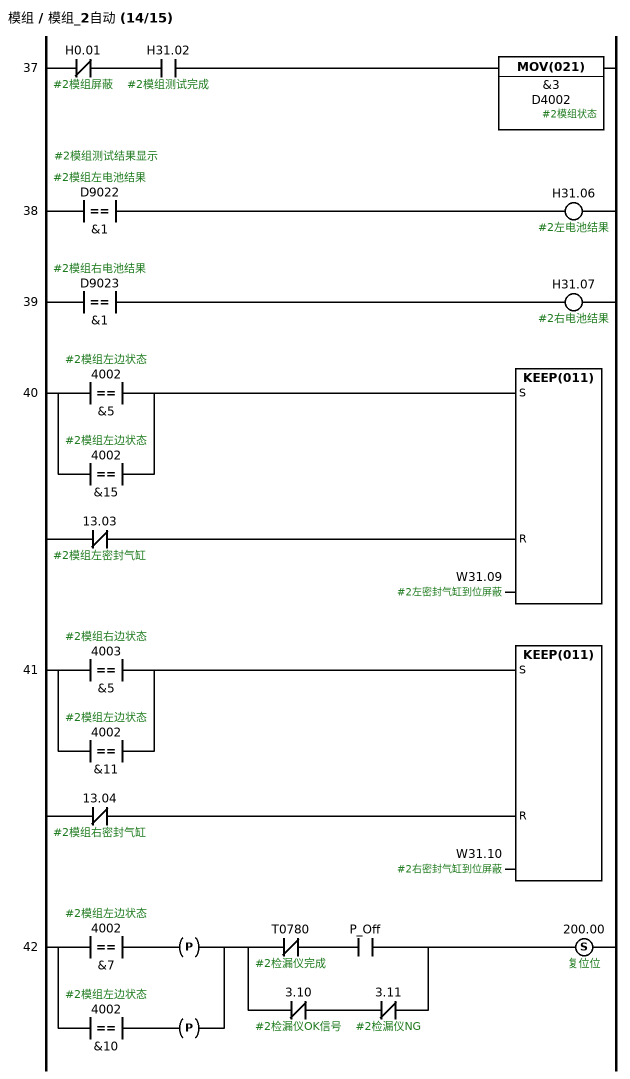
; [picture p233: 模组 / 模组_2自动, rungs 37-42]
; rung 37
LDNOT H0.01  ; #2模组屏蔽
AND H31.02  ; #2模组测试完成
MOV(021) &3 D4002  ; #2模组状态
; rung 38: #2模组测试结果显示
LD=(300) D9022 &1  ; #2模组左电池结果
OUT H31.06  ; #2左电池结果
; rung 39
LD=(300) D9023 &1  ; #2模组右电池结果
OUT H31.07  ; #2右电池结果
; rung 40
LD=(300) 4002 &5  ; #2模组左边状态
OR=(300) 4002 &15  ; #2模组左边状态
LDNOT 13.03  ; #2模组左密封气缸
KEEP(011) W31.09  ; #2左密封气缸到位屏蔽
; rung 41
LD=(300) 4003 &5  ; #2模组右边状态
OR=(300) 4002 &11  ; #2模组左边状态
LDNOT 13.04  ; #2模组右密封气缸
KEEP(011) W31.10  ; #2右密封气缸到位屏蔽
; rung 42
LD=(300) 4002 &7  ; #2模组左边状态
UP(521)
LD=(300) 4002 &10  ; #2模组左边状态
UP(521)
ORLD
LDNOT T0780  ; #2检漏仪完成
AND P_Off
LDNOT 3.10  ; #2检漏仪OK信号  // 2018/5/29hy修改,所有模组不在临抽气结束状态下，测试模组测试完成后，给出停止测试信号
ANDNOT 3.11  ; #2检漏仪NG
ORLD
ANDLD
SET 200.00  ; 复位位

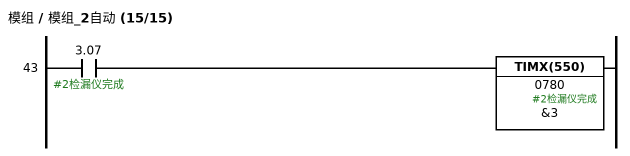
; rung 43
LD 3.07  ; #2检漏仪完成
TIMX(550) 0780 &3  ; #2检漏仪完成

### Section 模组_3自动

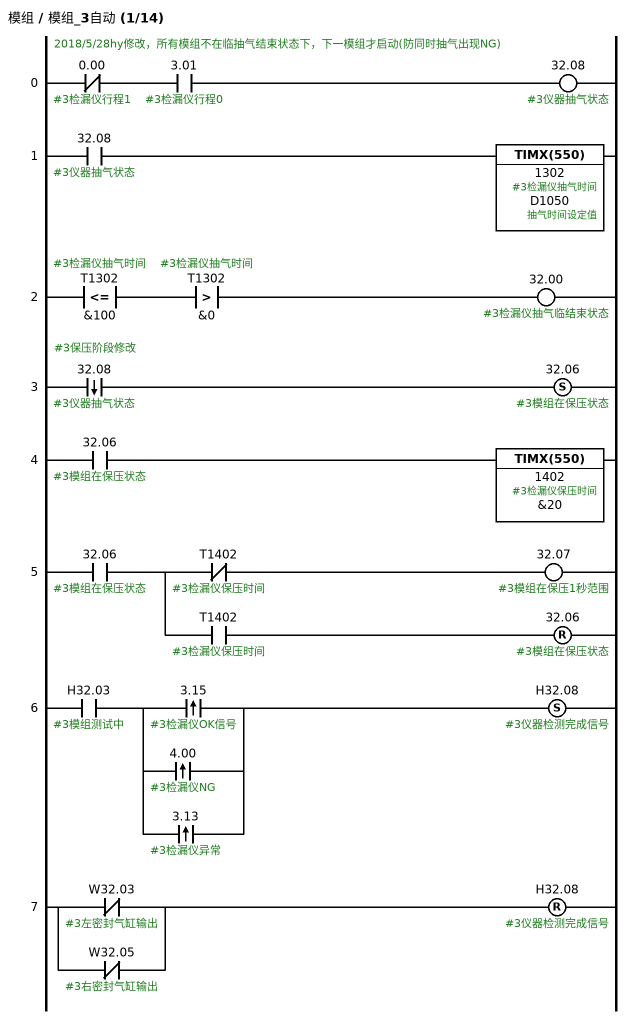
; rung 0: 2018/5/28hy修改，所有模组不在临抽气结束状态下，下一模组才启动(防同时抽气出现NG)
LDNOT 0.00  ; #3检漏仪行程1
AND 3.01  ; #3检漏仪行程0
OUT 32.08  ; #3仪器抽气状态
; rung 1
LD 32.08  ; #3仪器抽气状态
TIMX(550) 1302 D1050  ; 抽气时间设定值, #3检漏仪抽气时间
; rung 2
LD<=(315) T1302 &100  ; #3检漏仪抽气时间
AND>(320) T1302 &0  ; #3检漏仪抽气时间
OUT 32.00  ; #3检漏仪抽气临结束状态
; rung 3: #3保压阶段修改
%LD 32.08  ; #3仪器抽气状态
SET 32.06  ; #3模组在保压状态
; rung 4
LD 32.06  ; #3模组在保压状态
TIMX(550) 1402 &20  ; #3检漏仪保压时间
; rung 5
LD 32.06  ; #3模组在保压状态
OUT TR0
ANDNOT T1402  ; #3检漏仪保压时间
OUT 32.07  ; #3模组在保压1秒范围
LD TR0
AND T1402  ; #3检漏仪保压时间
RSET 32.06  ; #3模组在保压状态
; rung 6
LD H32.03  ; #3模组测试中
@LD 3.15  ; #3检漏仪OK信号
@OR 4.00  ; #3检漏仪NG
@OR 3.13  ; #3检漏仪异常
ANDLD
SET H32.08  ; #3仪器检测完成信号
; rung 7
LDNOT W32.03  ; #3左密封气缸输出
ORNOT W32.05  ; #3右密封气缸输出
RSET H32.08  ; #3仪器检测完成信号

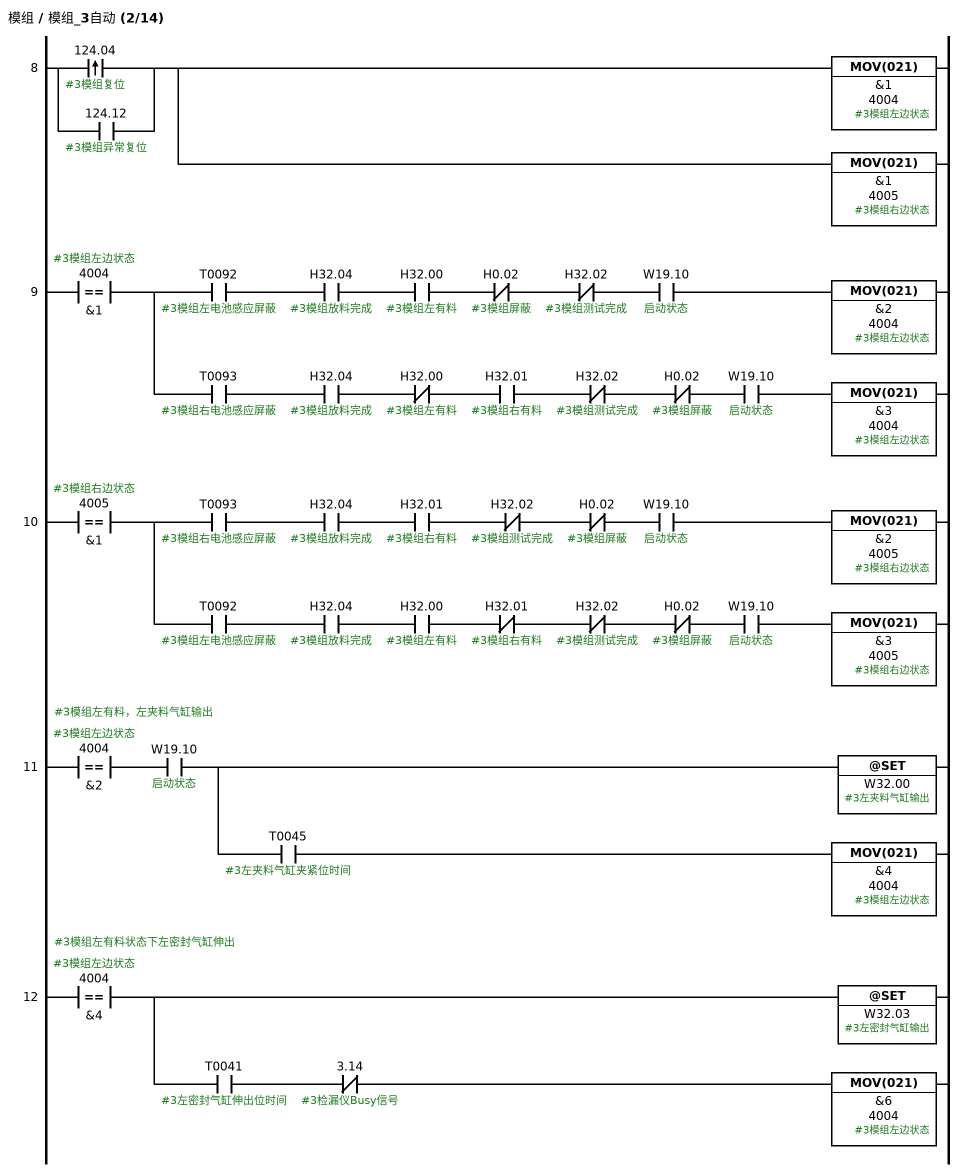
; rung 8
@LD 124.04  ; #3模组复位
OR 124.12  ; #3模组异常复位
MOV(021) &1 4004  ; #3模组左边状态
MOV(021) &1 4005  ; #3模组右边状态
; rung 9
LD=(300) 4004 &1  ; #3模组左边状态
OUT TR0
AND T0092  ; #3模组左电池感应屏蔽
AND H32.04  ; #3模组放料完成
AND H32.00  ; #3模组左有料
ANDNOT H0.02  ; #3模组屏蔽
ANDNOT H32.02  ; #3模组测试完成
AND W19.10  ; 启动状态
MOV(021) &2 4004  ; #3模组左边状态
LD TR0
AND T0093  ; #3模组右电池感应屏蔽
AND H32.04  ; #3模组放料完成
ANDNOT H32.00  ; #3模组左有料
AND H32.01  ; #3模组右有料
ANDNOT H32.02  ; #3模组测试完成
ANDNOT H0.02  ; #3模组屏蔽
AND W19.10  ; 启动状态
MOV(021) &3 4004  ; #3模组左边状态
; rung 10
LD=(300) 4005 &1  ; #3模组右边状态
OUT TR0
AND T0093  ; #3模组右电池感应屏蔽
AND H32.04  ; #3模组放料完成
AND H32.01  ; #3模组右有料
ANDNOT H32.02  ; #3模组测试完成
ANDNOT H0.02  ; #3模组屏蔽
AND W19.10  ; 启动状态
MOV(021) &2 4005  ; #3模组右边状态
LD TR0
AND T0092  ; #3模组左电池感应屏蔽
AND H32.04  ; #3模组放料完成
AND H32.00  ; #3模组左有料
ANDNOT H32.01  ; #3模组右有料
ANDNOT H32.02  ; #3模组测试完成
ANDNOT H0.02  ; #3模组屏蔽
AND W19.10  ; 启动状态
MOV(021) &3 4005  ; #3模组右边状态
; rung 11: #3模组左有料，左夹料气缸输出
LD=(300) 4004 &2  ; #3模组左边状态
AND W19.10  ; 启动状态
@SET W32.00  ; #3左夹料气缸输出
AND T0045  ; #3左夹料气缸夹紧位时间
MOV(021) &4 4004  ; #3模组左边状态
; rung 12: #3模组左有料状态下左密封气缸伸出
LD=(300) 4004 &4  ; #3模组左边状态
@SET W32.03  ; #3左密封气缸输出
AND T0041  ; #3左密封气缸伸出位时间
ANDNOT 3.14  ; #3检漏仪Busy信号
MOV(021) &6 4004  ; #3模组左边状态

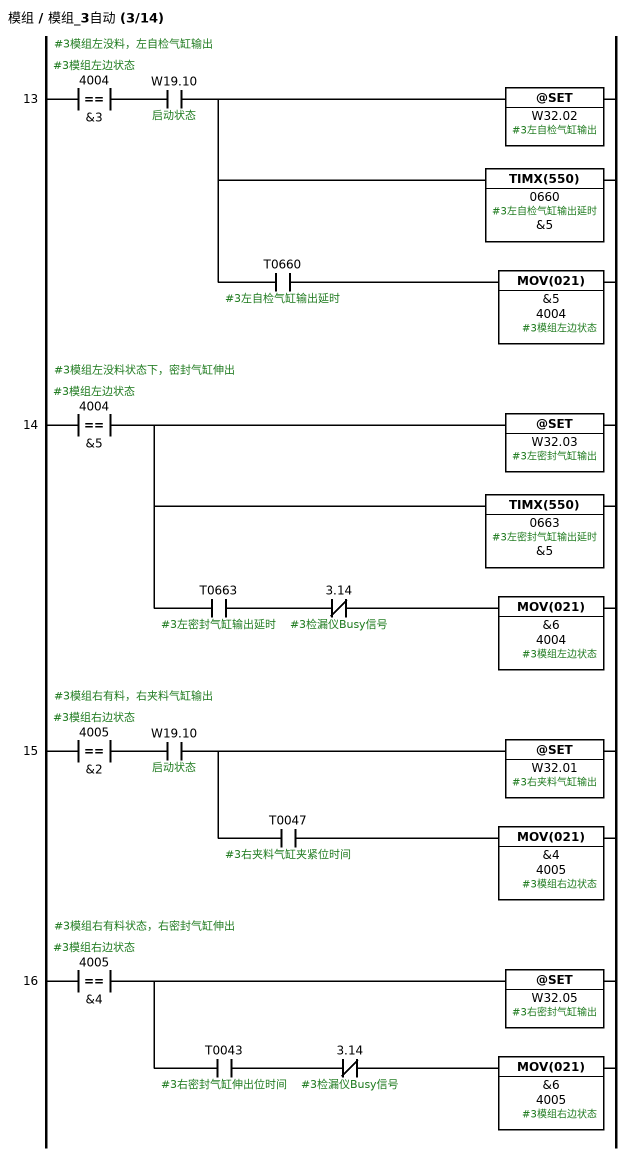
; rung 13: #3模组左没料，左自检气缸输出
LD=(300) 4004 &3  ; #3模组左边状态
AND W19.10  ; 启动状态
@SET W32.02  ; #3左自检气缸输出
TIMX(550) 0660 &5  ; #3左自检气缸输出延时
AND T0660  ; #3左自检气缸输出延时
MOV(021) &5 4004  ; #3模组左边状态
; rung 14: #3模组左没料状态下，密封气缸伸出
LD=(300) 4004 &5  ; #3模组左边状态
@SET W32.03  ; #3左密封气缸输出
TIMX(550) 0663 &5  ; #3左密封气缸输出延时
AND T0663  ; #3左密封气缸输出延时
ANDNOT 3.14  ; #3检漏仪Busy信号
MOV(021) &6 4004  ; #3模组左边状态
; rung 15: #3模组右有料，右夹料气缸输出
LD=(300) 4005 &2  ; #3模组右边状态
AND W19.10  ; 启动状态
@SET W32.01  ; #3右夹料气缸输出
AND T0047  ; #3右夹料气缸夹紧位时间
MOV(021) &4 4005  ; #3模组右边状态
; rung 16: #3模组右有料状态，右密封气缸伸出
LD=(300) 4005 &4  ; #3模组右边状态
@SET W32.05  ; #3右密封气缸输出
AND T0043  ; #3右密封气缸伸出位时间
ANDNOT 3.14  ; #3检漏仪Busy信号
MOV(021) &6 4005  ; #3模组右边状态

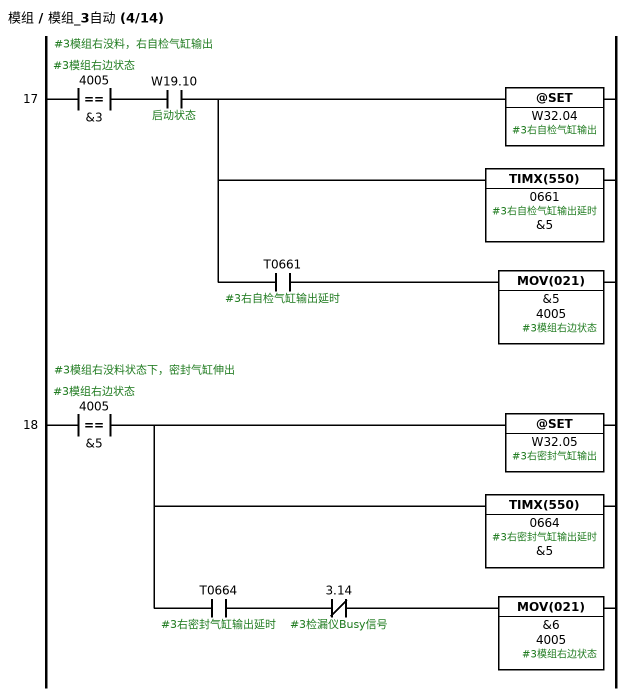
; rung 17: #3模组右没料，右自检气缸输出
LD=(300) 4005 &3  ; #3模组右边状态
AND W19.10  ; 启动状态
@SET W32.04  ; #3右自检气缸输出
TIMX(550) 0661 &5  ; #3右自检气缸输出延时
AND T0661  ; #3右自检气缸输出延时
MOV(021) &5 4005  ; #3模组右边状态
; rung 18: #3模组右没料状态下，密封气缸伸出
LD=(300) 4005 &5  ; #3模组右边状态
@SET W32.05  ; #3右密封气缸输出
TIMX(550) 0664 &5  ; #3右密封气缸输出延时
AND T0664  ; #3右密封气缸输出延时
ANDNOT 3.14  ; #3检漏仪Busy信号
MOV(021) &6 4005  ; #3模组右边状态

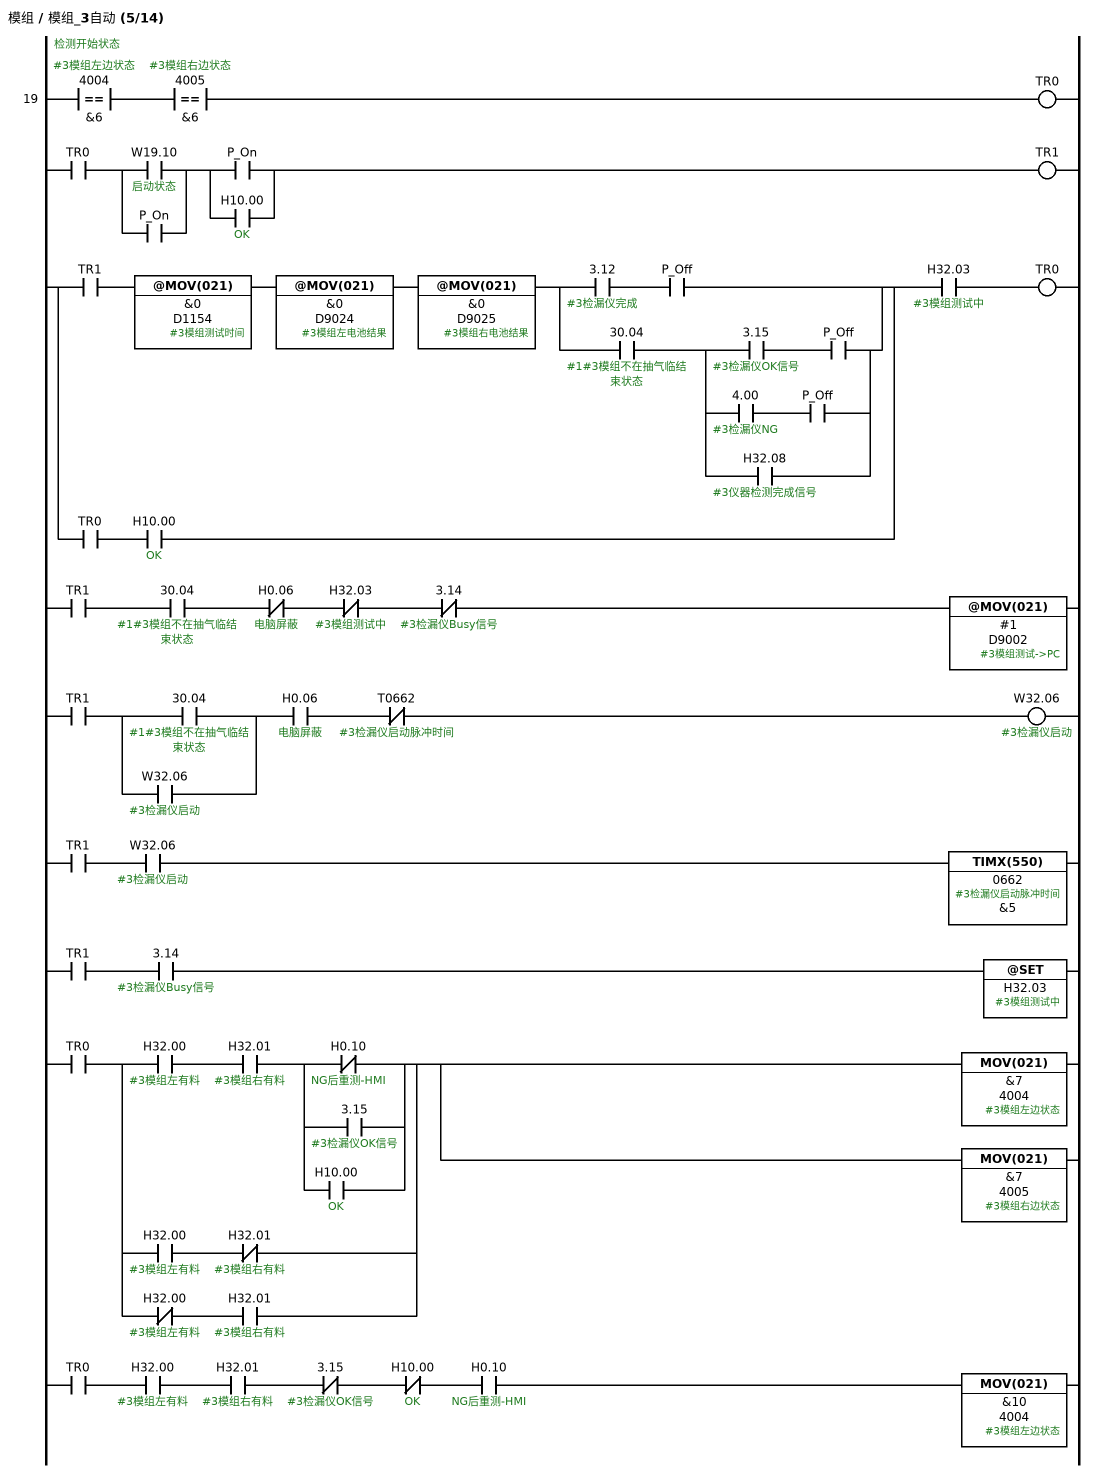
; rung 19: 检测开始状态
LD=(300) 4004 &6  ; #3模组左边状态
AND=(300) 4005 &6  ; #3模组右边状态
OUT TR0
LD W19.10  ; 启动状态
OR P_On
ANDLD
LD P_On  // 2018/5/28hy修改 所有模组不在抽气临结束状态下，下一模组才能启动(防抽气NG)
OR H10.00  ; OK
ANDLD
OUT TR1
AND 30.04  ; #1#3模组不在抽气临结束状态  // 2018/5/28hy修改 所有模组不在抽气临结束状态下，下一模组才能启动(防抽气NG)
ANDNOT H0.06  ; 电脑屏蔽
ANDNOT H32.03  ; #3模组测试中
ANDNOT 3.14  ; #3检漏仪Busy信号
@MOV(021) #1 D9002  ; #3模组测试->PC
LD TR1
LD 30.04  ; #1#3模组不在抽气临结束状态  // 2018/5/28hy修改 所有模组不在抽气临结束状态下，下一模组才能启动(防抽气NG)
OR W32.06  ; #3检漏仪启动
ANDLD
AND H0.06  ; 电脑屏蔽
ANDNOT T0662  ; #3检漏仪启动脉冲时间
OUT W32.06  ; #3检漏仪启动
LD TR1
AND W32.06  ; #3检漏仪启动
TIMX(550) 0662 &5  ; #3检漏仪启动脉冲时间
LD TR1
AND 3.14  ; #3检漏仪Busy信号
@SET H32.03  ; #3模组测试中
LD TR1
@MOV(021) &0 D1154  ; #3模组测试时间
@MOV(021) &0 D9024  ; #3模组左电池结果
@MOV(021) &0 D9025  ; #3模组右电池结果
LD 3.12  ; #3检漏仪完成
AND P_Off
LD 30.04  ; #1#3模组不在抽气临结束状态  // 2018/5/29hy修改,所有模组不在临抽气结束状态下，测试模组测试完成后，给出停止测试信号
LD 3.15  ; #3检漏仪OK信号
AND P_Off
LD 4.00  ; #3检漏仪NG
AND P_Off
ORLD
OR H32.08  ; #3仪器检测完成信号
ANDLD
ORLD
ANDLD
LD TR0
AND H10.00  ; OK
ORLD
AND H32.03  ; #3模组测试中
OUT TR0
LD H32.00  ; #3模组左有料
AND H32.01  ; #3模组右有料
LDNOT H0.10  ; NG后重测-HMI
OR 3.15  ; #3检漏仪OK信号
OR H10.00  ; OK
ANDLD
LD H32.00  ; #3模组左有料
ANDNOT H32.01  ; #3模组右有料
ORLD
LDNOT H32.00  ; #3模组左有料
AND H32.01  ; #3模组右有料
ORLD
ANDLD
MOV(021) &7 4004  ; #3模组左边状态
MOV(021) &7 4005  ; #3模组右边状态
LD TR0
AND H32.00  ; #3模组左有料
AND H32.01  ; #3模组右有料
ANDNOT 3.15  ; #3检漏仪OK信号
ANDNOT H10.00  ; OK
AND H0.10  ; NG后重测-HMI
MOV(021) &10 4004  ; #3模组左边状态

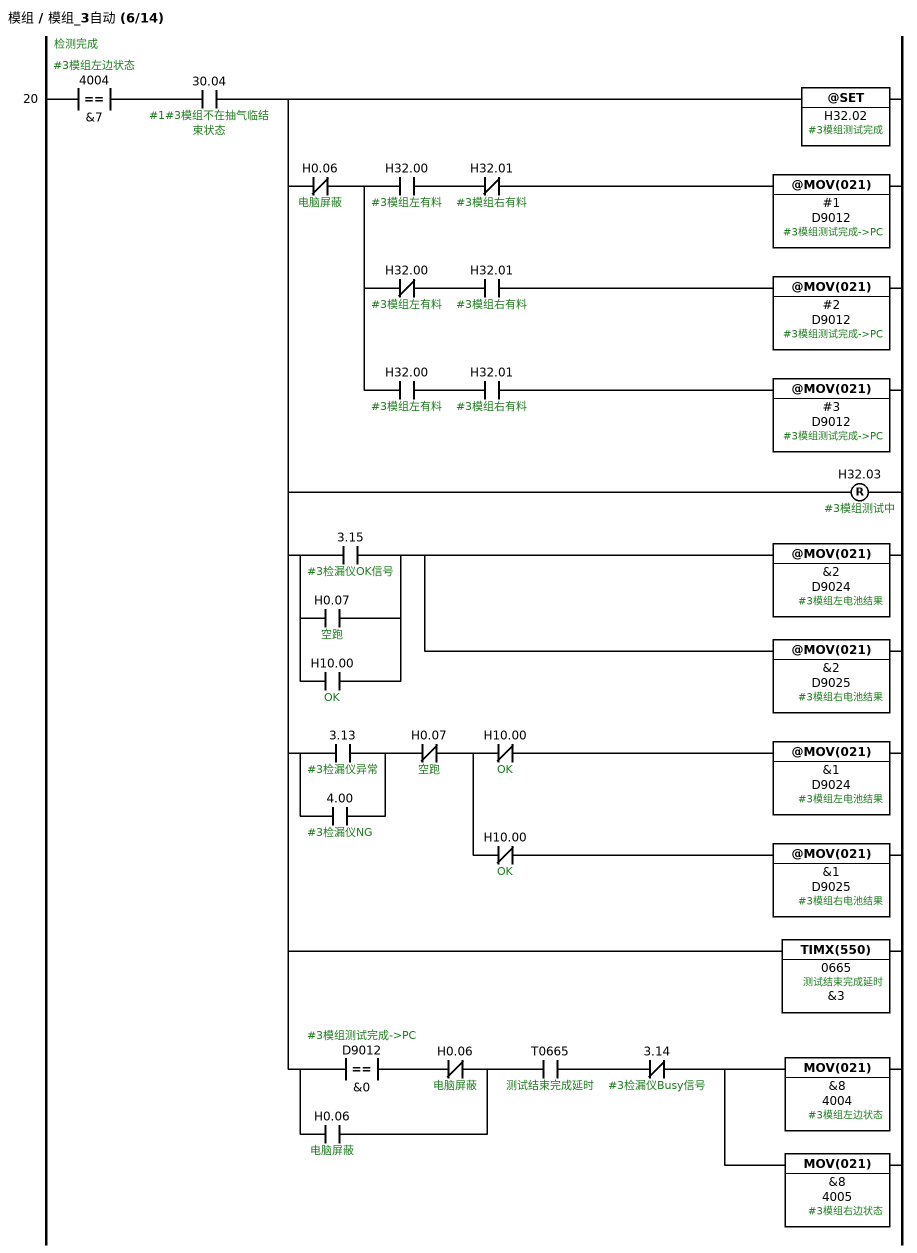
; rung 20: 检测完成
LD=(300) 4004 &7  ; #3模组左边状态
AND 30.04  ; #1#3模组不在抽气临结束状态
OUT TR0
@SET H32.02  ; #3模组测试完成
ANDNOT H0.06  ; 电脑屏蔽
OUT TR1
AND H32.00  ; #3模组左有料
ANDNOT H32.01  ; #3模组右有料
@MOV(021) #1 D9012  ; #3模组测试完成->PC
LD TR1
ANDNOT H32.00  ; #3模组左有料
AND H32.01  ; #3模组右有料
@MOV(021) #2 D9012  ; #3模组测试完成->PC
LD TR1
AND H32.00  ; #3模组左有料
AND H32.01  ; #3模组右有料
@MOV(021) #3 D9012  ; #3模组测试完成->PC
LD TR0
RSET H32.03  ; #3模组测试中
LD 3.15  ; #3检漏仪OK信号
OR H0.07  ; 空跑
OR H10.00  ; OK
ANDLD
@MOV(021) &2 D9024  ; #3模组左电池结果
@MOV(021) &2 D9025  ; #3模组右电池结果
LD TR0
LD 3.13  ; #3检漏仪异常
OR 4.00  ; #3检漏仪NG
ANDLD
ANDNOT H0.07  ; 空跑
OUT TR1
ANDNOT H10.00  ; OK
@MOV(021) &1 D9024  ; #3模组左电池结果
LD TR1
ANDNOT H10.00  ; OK
@MOV(021) &1 D9025  ; #3模组右电池结果
LD TR0
TIMX(550) 0665 &3  ; 测试结束完成延时
LD=(300) D9012 &0  ; #3模组测试完成->PC
ANDNOT H0.06  ; 电脑屏蔽
OR H0.06  ; 电脑屏蔽
ANDLD
AND T0665  ; 测试结束完成延时
ANDNOT 3.14  ; #3检漏仪Busy信号
MOV(021) &8 4004  ; #3模组左边状态
MOV(021) &8 4005  ; #3模组右边状态

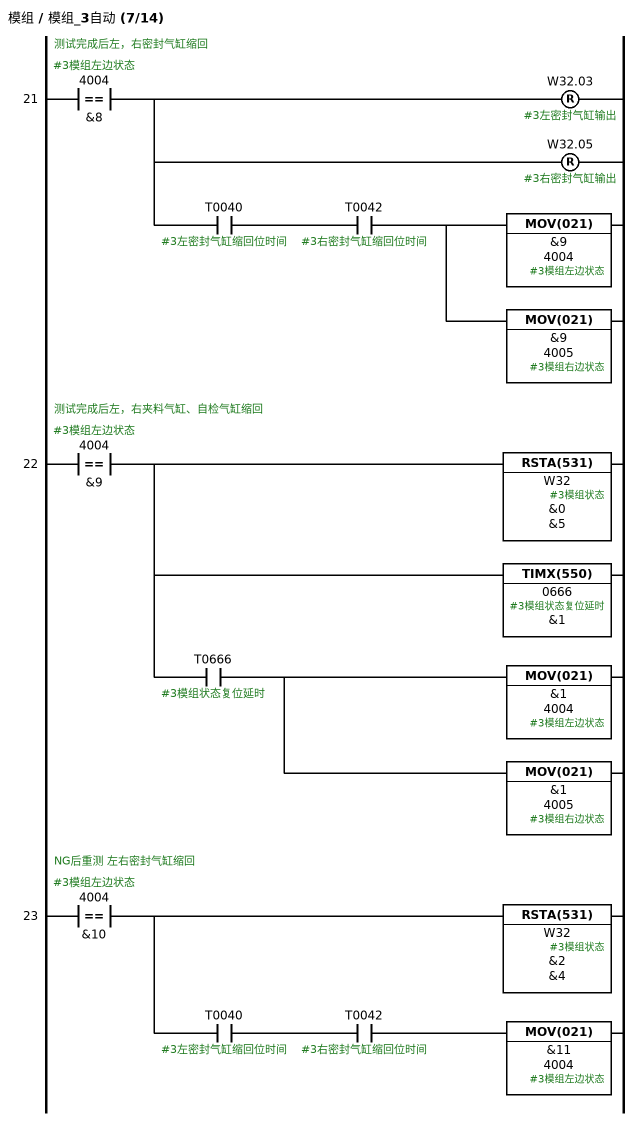
; rung 21: 测试完成后左，右密封气缸缩回
LD=(300) 4004 &8  ; #3模组左边状态
RSET W32.03  ; #3左密封气缸输出
RSET W32.05  ; #3右密封气缸输出
AND T0040  ; #3左密封气缸缩回位时间
AND T0042  ; #3右密封气缸缩回位时间
MOV(021) &9 4004  ; #3模组左边状态
MOV(021) &9 4005  ; #3模组右边状态
; rung 22: 测试完成后左，右夹料气缸、自检气缸缩回
LD=(300) 4004 &9  ; #3模组左边状态
RSTA(531) W32 &0 &5  ; #3模组状态
TIMX(550) 0666 &1  ; #3模组状态复位延时
AND T0666  ; #3模组状态复位延时
MOV(021) &1 4004  ; #3模组左边状态
MOV(021) &1 4005  ; #3模组右边状态
; rung 23: NG后重测 左右密封气缸缩回
LD=(300) 4004 &10  ; #3模组左边状态
RSTA(531) W32 &2 &4  ; #3模组状态
AND T0040  ; #3左密封气缸缩回位时间
AND T0042  ; #3右密封气缸缩回位时间
MOV(021) &11 4004  ; #3模组左边状态

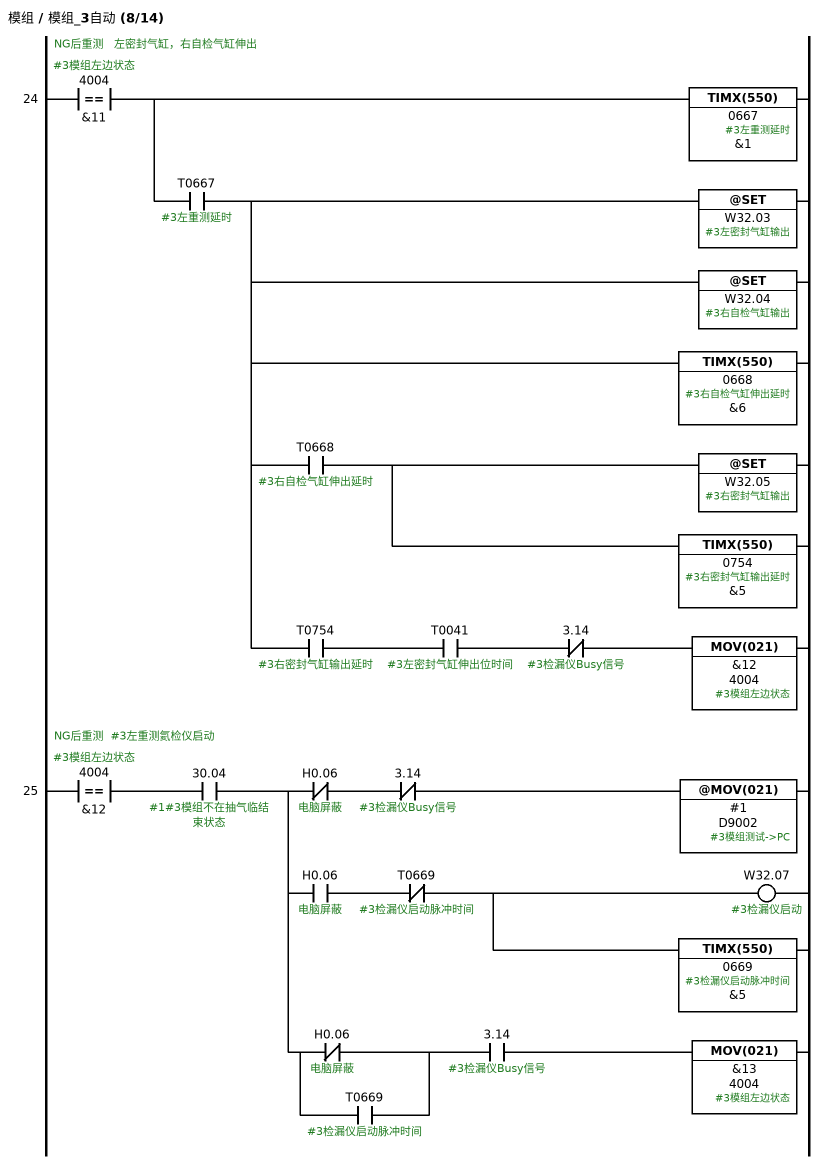
; rung 24: NG后重测   左密封气缸，右自检气缸伸出
LD=(300) 4004 &11  ; #3模组左边状态
TIMX(550) 0667 &1  ; #3左重测延时
AND T0667  ; #3左重测延时
OUT TR0
@SET W32.03  ; #3左密封气缸输出
@SET W32.04  ; #3右自检气缸输出
TIMX(550) 0668 &6  ; #3右自检气缸伸出延时
AND T0668  ; #3右自检气缸伸出延时
@SET W32.05  ; #3右密封气缸输出
TIMX(550) 0754 &5  ; #3右密封气缸输出延时
LD TR0
AND T0754  ; #3右密封气缸输出延时
AND T0041  ; #3左密封气缸伸出位时间
ANDNOT 3.14  ; #3检漏仪Busy信号
MOV(021) &12 4004  ; #3模组左边状态
; rung 25: NG后重测  #3左重测氦检仪启动
LD=(300) 4004 &12  ; #3模组左边状态
AND 30.04  ; #1#3模组不在抽气临结束状态  // 2018/5/28hy修改 所有模组不在抽气临结束状态下，下一模组才能启动(防抽气NG)
OUT TR0
ANDNOT H0.06  ; 电脑屏蔽
ANDNOT 3.14  ; #3检漏仪Busy信号
@MOV(021) #1 D9002  ; #3模组测试->PC
LD TR0
AND H0.06  ; 电脑屏蔽
ANDNOT T0669  ; #3检漏仪启动脉冲时间
OUT W32.07  ; #3检漏仪启动
TIMX(550) 0669 &5  ; #3检漏仪启动脉冲时间
LD TR0
LDNOT H0.06  ; 电脑屏蔽
OR T0669  ; #3检漏仪启动脉冲时间
ANDLD
AND 3.14  ; #3检漏仪Busy信号
MOV(021) &13 4004  ; #3模组左边状态

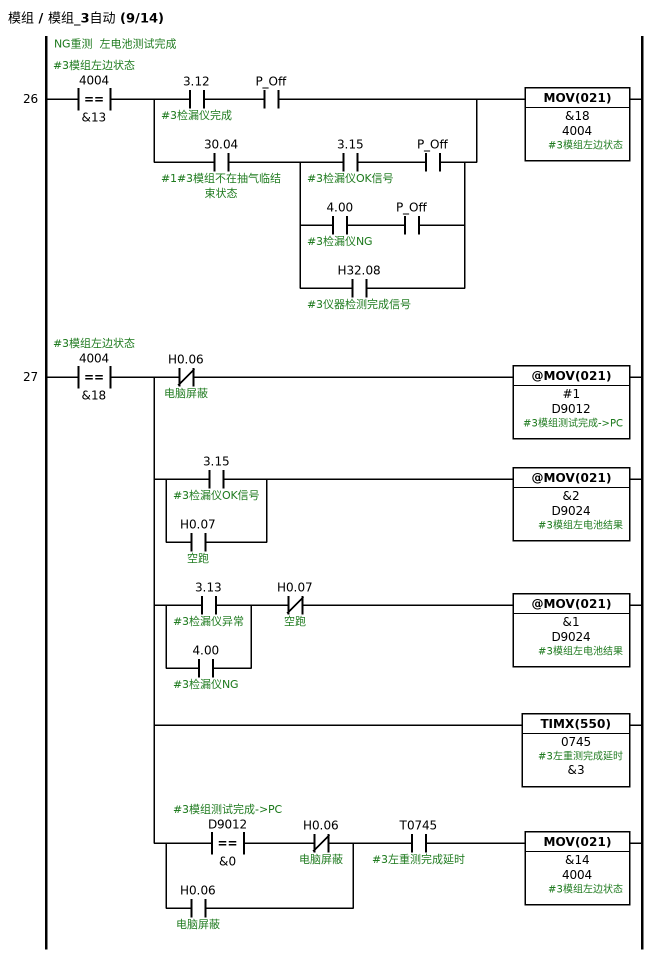
; rung 26: NG重测  左电池测试完成
LD=(300) 4004 &13  ; #3模组左边状态
LD 3.12  ; #3检漏仪完成
AND P_Off
LD 30.04  ; #1#3模组不在抽气临结束状态  // 2018/5/29hy修改,所有模组不在临抽气结束状态下，测试模组测试完成后，给出停止测试信号
LD 3.15  ; #3检漏仪OK信号
AND P_Off
LD 4.00  ; #3检漏仪NG
AND P_Off
ORLD
OR H32.08  ; #3仪器检测完成信号
ANDLD
ORLD
ANDLD
MOV(021) &18 4004  ; #3模组左边状态
; rung 27
LD=(300) 4004 &18  ; #3模组左边状态
OUT TR0
ANDNOT H0.06  ; 电脑屏蔽
@MOV(021) #1 D9012  ; #3模组测试完成->PC
LD TR0
LD 3.15  ; #3检漏仪OK信号
OR H0.07  ; 空跑
ANDLD
@MOV(021) &2 D9024  ; #3模组左电池结果
LD TR0
LD 3.13  ; #3检漏仪异常
OR 4.00  ; #3检漏仪NG
ANDLD
ANDNOT H0.07  ; 空跑
@MOV(021) &1 D9024  ; #3模组左电池结果
LD TR0
TIMX(550) 0745 &3  ; #3左重测完成延时
LD=(300) D9012 &0  ; #3模组测试完成->PC
ANDNOT H0.06  ; 电脑屏蔽
OR H0.06  ; 电脑屏蔽
ANDLD
AND T0745  ; #3左重测完成延时
MOV(021) &14 4004  ; #3模组左边状态

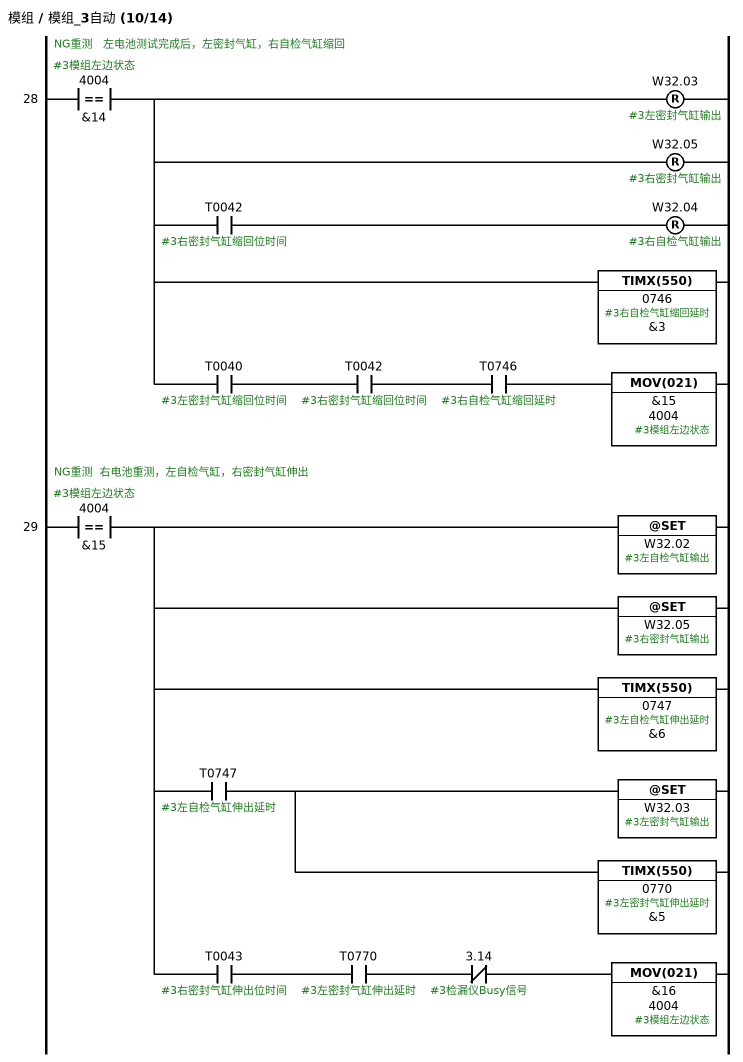
; rung 28: NG重测   左电池测试完成后，左密封气缸，右自检气缸缩回
LD=(300) 4004 &14  ; #3模组左边状态
OUT TR0
RSET W32.03  ; #3左密封气缸输出
RSET W32.05  ; #3右密封气缸输出
AND T0042  ; #3右密封气缸缩回位时间
RSET W32.04  ; #3右自检气缸输出
LD TR0
TIMX(550) 0746 &3  ; #3右自检气缸缩回延时
AND T0040  ; #3左密封气缸缩回位时间
AND T0042  ; #3右密封气缸缩回位时间
AND T0746  ; #3右自检气缸缩回延时
MOV(021) &15 4004  ; #3模组左边状态
; rung 29: NG重测  右电池重测，左自检气缸，右密封气缸伸出
LD=(300) 4004 &15  ; #3模组左边状态
OUT TR0
@SET W32.02  ; #3左自检气缸输出
@SET W32.05  ; #3右密封气缸输出
TIMX(550) 0747 &6  ; #3左自检气缸伸出延时
AND T0747  ; #3左自检气缸伸出延时
@SET W32.03  ; #3左密封气缸输出
TIMX(550) 0770 &5  ; #3左密封气缸伸出延时
LD TR0
AND T0043  ; #3右密封气缸伸出位时间
AND T0770  ; #3左密封气缸伸出延时
ANDNOT 3.14  ; #3检漏仪Busy信号
MOV(021) &16 4004  ; #3模组左边状态

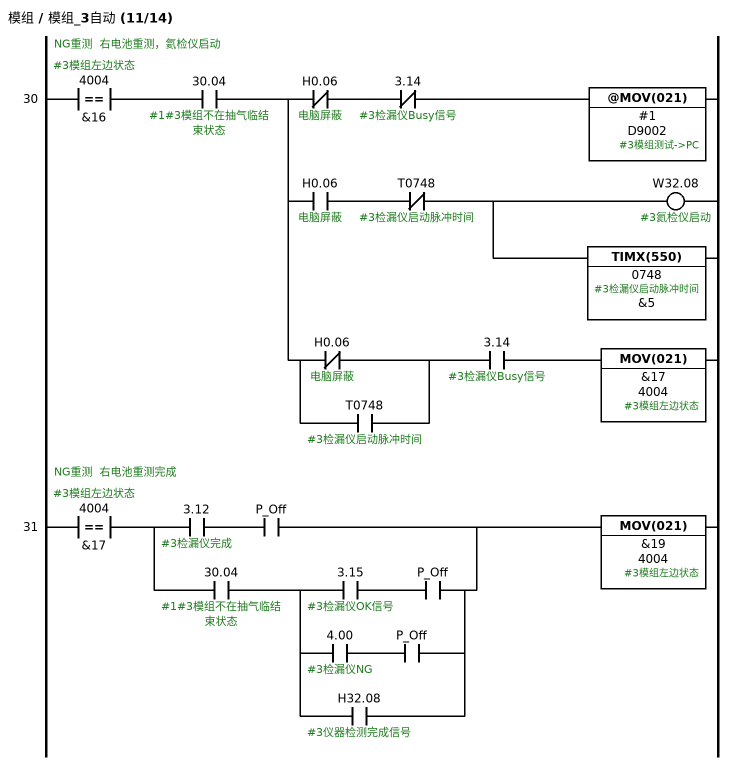
; rung 30: NG重测  右电池重测，氦检仪启动
LD=(300) 4004 &16  ; #3模组左边状态
AND 30.04  ; #1#3模组不在抽气临结束状态  // 2018/5/28hy修改 所有模组不在抽气临结束状态下，下一模组才能启动(防抽气NG)
OUT TR0
ANDNOT H0.06  ; 电脑屏蔽
ANDNOT 3.14  ; #3检漏仪Busy信号
@MOV(021) #1 D9002  ; #3模组测试->PC
LD TR0
AND H0.06  ; 电脑屏蔽
ANDNOT T0748  ; #3检漏仪启动脉冲时间
OUT W32.08  ; #3氦检仪启动
TIMX(550) 0748 &5  ; #3检漏仪启动脉冲时间
LD TR0
LDNOT H0.06  ; 电脑屏蔽
OR T0748  ; #3检漏仪启动脉冲时间
ANDLD
AND 3.14  ; #3检漏仪Busy信号
MOV(021) &17 4004  ; #3模组左边状态
; rung 31: NG重测  右电池重测完成
LD=(300) 4004 &17  ; #3模组左边状态
LD 3.12  ; #3检漏仪完成
AND P_Off
LD 30.04  ; #1#3模组不在抽气临结束状态  // 2018/5/29hy修改,所有模组不在临抽气结束状态下，测试模组测试完成后，给出停止测试信号
LD 3.15  ; #3检漏仪OK信号
AND P_Off
LD 4.00  ; #3检漏仪NG
AND P_Off
ORLD
OR H32.08  ; #3仪器检测完成信号
ANDLD
ORLD
ANDLD
MOV(021) &19 4004  ; #3模组左边状态

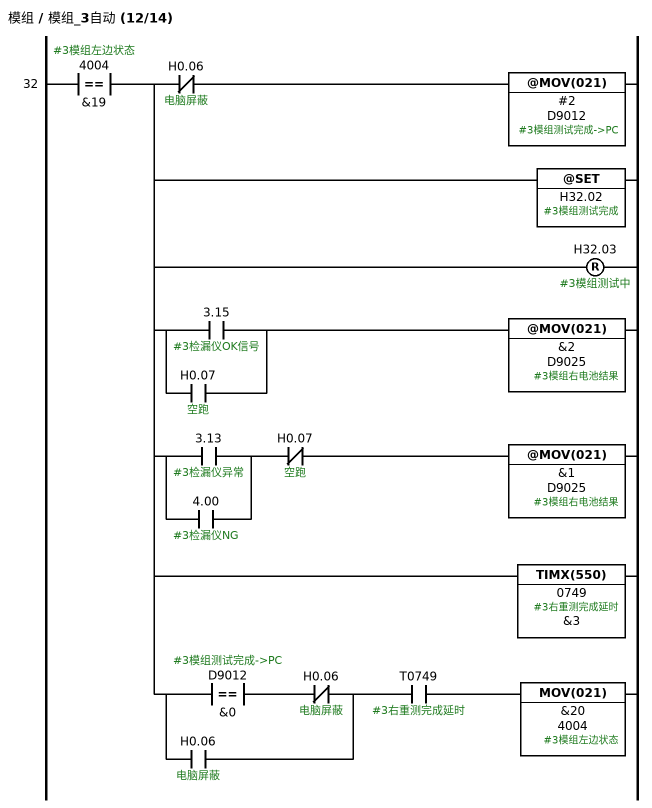
; rung 32
LD=(300) 4004 &19  ; #3模组左边状态
OUT TR0
ANDNOT H0.06  ; 电脑屏蔽
@MOV(021) #2 D9012  ; #3模组测试完成->PC
LD TR0
@SET H32.02  ; #3模组测试完成
RSET H32.03  ; #3模组测试中
LD 3.15  ; #3检漏仪OK信号
OR H0.07  ; 空跑
ANDLD
@MOV(021) &2 D9025  ; #3模组右电池结果
LD TR0
LD 3.13  ; #3检漏仪异常
OR 4.00  ; #3检漏仪NG
ANDLD
ANDNOT H0.07  ; 空跑
@MOV(021) &1 D9025  ; #3模组右电池结果
LD TR0
TIMX(550) 0749 &3  ; #3右重测完成延时
LD=(300) D9012 &0  ; #3模组测试完成->PC
ANDNOT H0.06  ; 电脑屏蔽
OR H0.06  ; 电脑屏蔽
ANDLD
AND T0749  ; #3右重测完成延时
MOV(021) &20 4004  ; #3模组左边状态

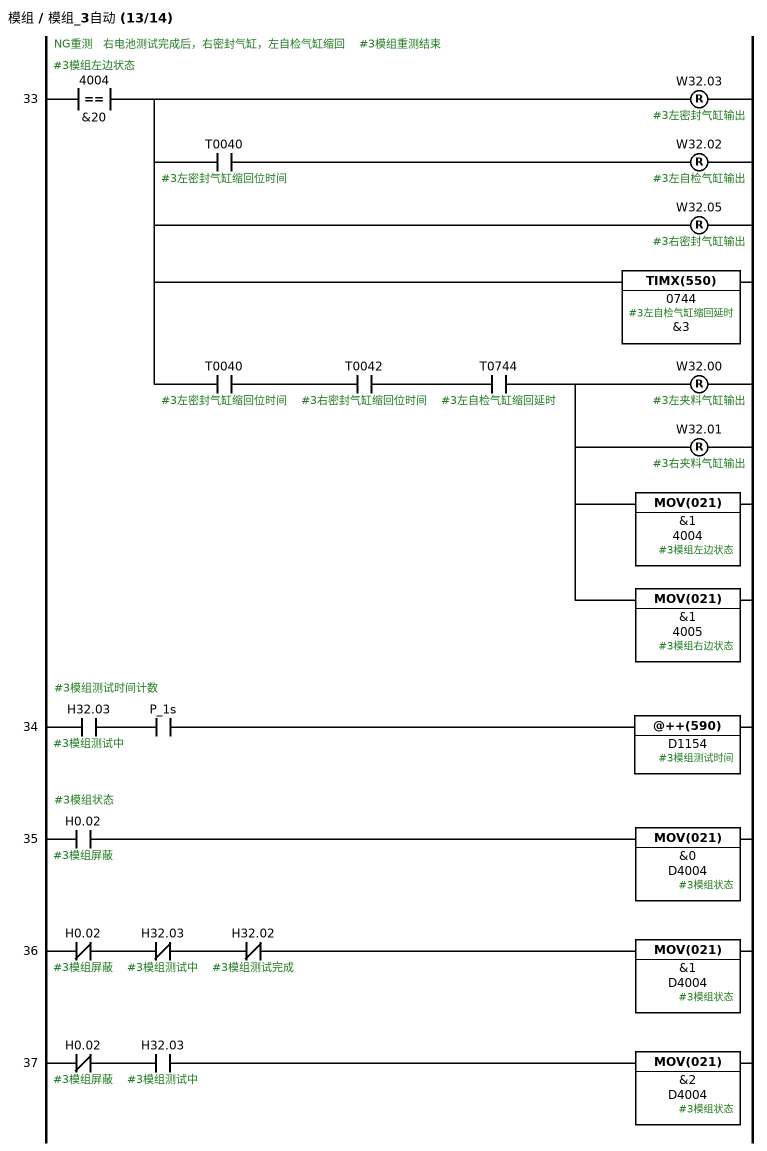
; rung 33: NG重测   右电池测试完成后，右密封气缸，左自检气缸缩回    #3模组重测结束
LD=(300) 4004 &20  ; #3模组左边状态
OUT TR0
RSET W32.03  ; #3左密封气缸输出
AND T0040  ; #3左密封气缸缩回位时间
RSET W32.02  ; #3左自检气缸输出
LD TR0
RSET W32.05  ; #3右密封气缸输出
TIMX(550) 0744 &3  ; #3左自检气缸缩回延时
AND T0040  ; #3左密封气缸缩回位时间
AND T0042  ; #3右密封气缸缩回位时间
AND T0744  ; #3左自检气缸缩回延时
RSET W32.00  ; #3左夹料气缸输出
RSET W32.01  ; #3右夹料气缸输出
MOV(021) &1 4004  ; #3模组左边状态
MOV(021) &1 4005  ; #3模组右边状态
; rung 34: #3模组测试时间计数
LD H32.03  ; #3模组测试中
AND P_1s
@++(590) D1154  ; #3模组测试时间
; rung 35: #3模组状态
LD H0.02  ; #3模组屏蔽
MOV(021) &0 D4004  ; #3模组状态
; rung 36
LDNOT H0.02  ; #3模组屏蔽
ANDNOT H32.03  ; #3模组测试中
ANDNOT H32.02  ; #3模组测试完成
MOV(021) &1 D4004  ; #3模组状态
; rung 37
LDNOT H0.02  ; #3模组屏蔽
AND H32.03  ; #3模组测试中
MOV(021) &2 D4004  ; #3模组状态

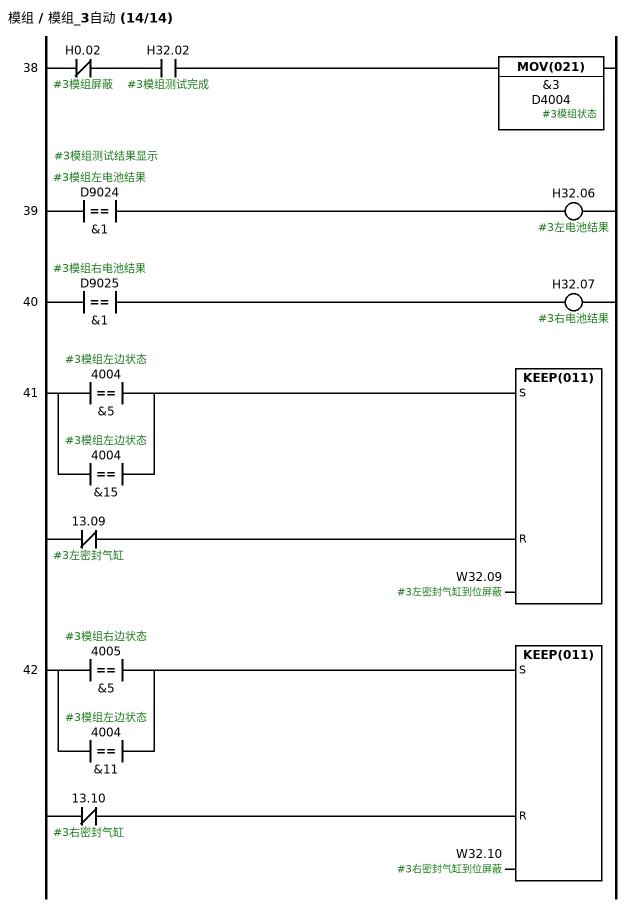
; rung 38
LDNOT H0.02  ; #3模组屏蔽
AND H32.02  ; #3模组测试完成
MOV(021) &3 D4004  ; #3模组状态
; rung 39: #3模组测试结果显示
LD=(300) D9024 &1  ; #3模组左电池结果
OUT H32.06  ; #3左电池结果
; rung 40
LD=(300) D9025 &1  ; #3模组右电池结果
OUT H32.07  ; #3右电池结果
; rung 41
LD=(300) 4004 &5  ; #3模组左边状态
OR=(300) 4004 &15  ; #3模组左边状态
LDNOT 13.09  ; #3左密封气缸
KEEP(011) W32.09  ; #3左密封气缸到位屏蔽
; rung 42
LD=(300) 4005 &5  ; #3模组右边状态
OR=(300) 4004 &11  ; #3模组左边状态
LDNOT 13.10  ; #3右密封气缸
KEEP(011) W32.10  ; #3右密封气缸到位屏蔽

### Section 模组_4自动

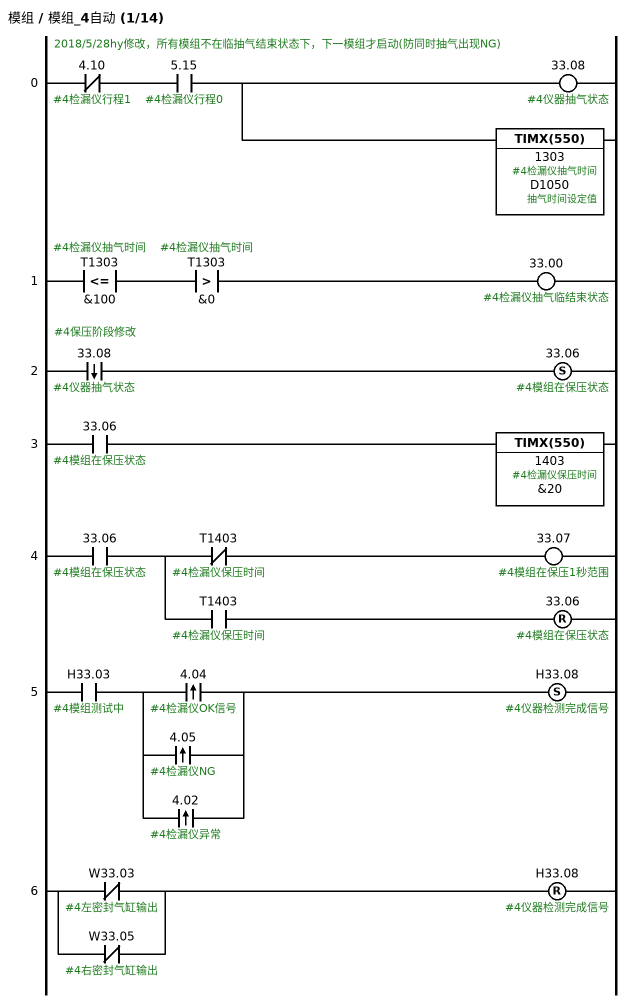
; rung 0: 2018/5/28hy修改，所有模组不在临抽气结束状态下，下一模组才启动(防同时抽气出现NG)
LDNOT 4.10  ; #4检漏仪行程1
AND 5.15  ; #4检漏仪行程0
OUT 33.08  ; #4仪器抽气状态
TIMX(550) 1303 D1050  ; 抽气时间设定值, #4检漏仪抽气时间
; rung 1
LD<=(315) T1303 &100  ; #4检漏仪抽气时间
AND>(320) T1303 &0  ; #4检漏仪抽气时间
OUT 33.00  ; #4检漏仪抽气临结束状态
; rung 2: #4保压阶段修改
%LD 33.08  ; #4仪器抽气状态
SET 33.06  ; #4模组在保压状态
; rung 3
LD 33.06  ; #4模组在保压状态
TIMX(550) 1403 &20  ; #4检漏仪保压时间
; rung 4
LD 33.06  ; #4模组在保压状态
OUT TR0
ANDNOT T1403  ; #4检漏仪保压时间
OUT 33.07  ; #4模组在保压1秒范围
LD TR0
AND T1403  ; #4检漏仪保压时间
RSET 33.06  ; #4模组在保压状态
; rung 5
LD H33.03  ; #4模组测试中
@LD 4.04  ; #4检漏仪OK信号
@OR 4.05  ; #4检漏仪NG
@OR 4.02  ; #4检漏仪异常
ANDLD
SET H33.08  ; #4仪器检测完成信号
; rung 6
LDNOT W33.03  ; #4左密封气缸输出
ORNOT W33.05  ; #4右密封气缸输出
RSET H33.08  ; #4仪器检测完成信号

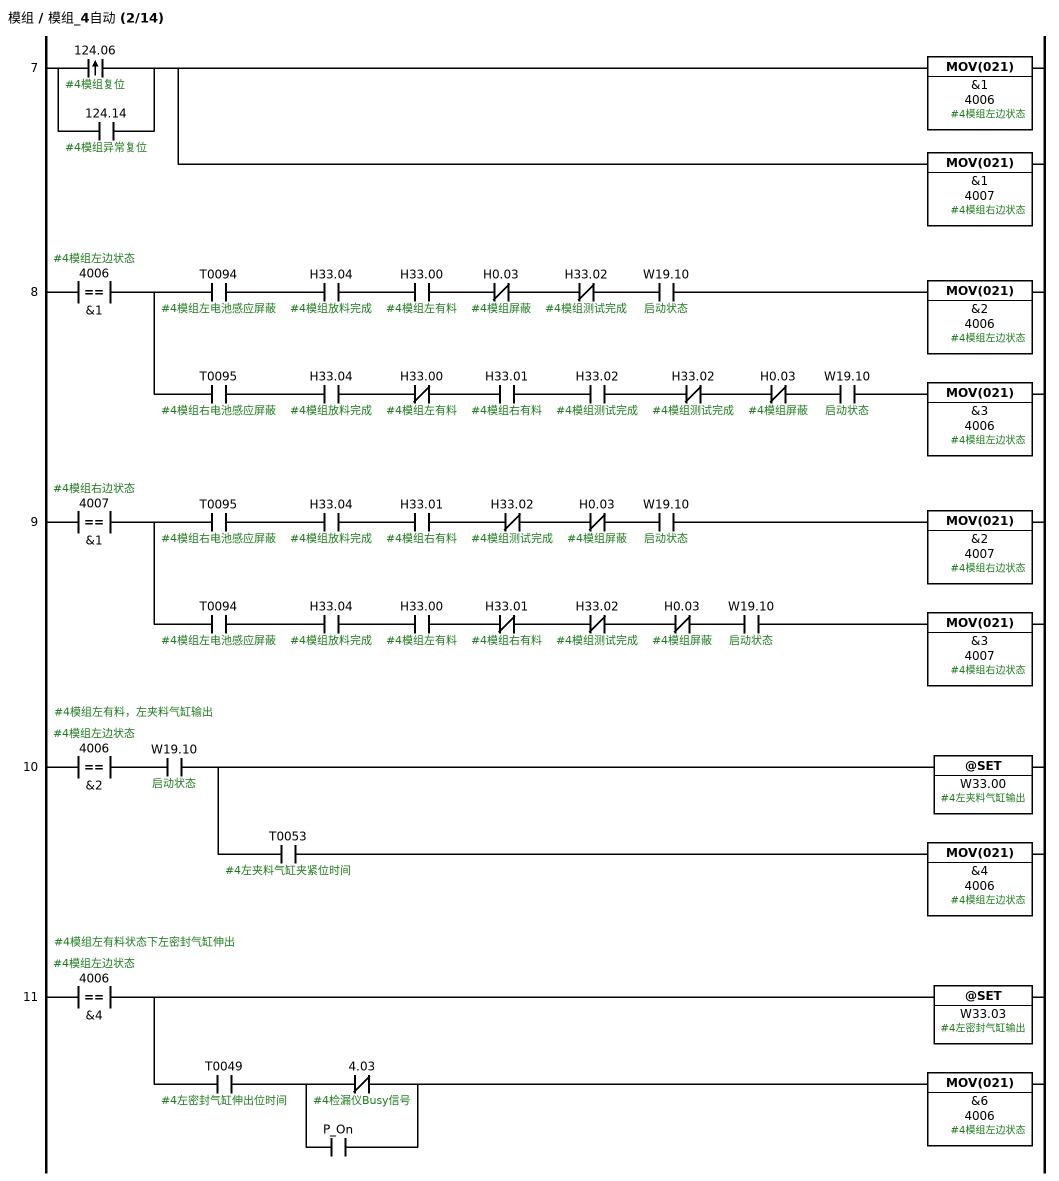
; rung 7
@LD 124.06  ; #4模组复位
OR 124.14  ; #4模组异常复位
MOV(021) &1 4006  ; #4模组左边状态
MOV(021) &1 4007  ; #4模组右边状态
; rung 8
LD=(300) 4006 &1  ; #4模组左边状态
OUT TR0
AND T0094  ; #4模组左电池感应屏蔽
AND H33.04  ; #4模组放料完成
AND H33.00  ; #4模组左有料
ANDNOT H0.03  ; #4模组屏蔽
ANDNOT H33.02  ; #4模组测试完成
AND W19.10  ; 启动状态
MOV(021) &2 4006  ; #4模组左边状态
LD TR0
AND T0095  ; #4模组右电池感应屏蔽
AND H33.04  ; #4模组放料完成
ANDNOT H33.00  ; #4模组左有料
AND H33.01  ; #4模组右有料
AND H33.02  ; #4模组测试完成
ANDNOT H33.02  ; #4模组测试完成
ANDNOT H0.03  ; #4模组屏蔽
AND W19.10  ; 启动状态
MOV(021) &3 4006  ; #4模组左边状态
; rung 9
LD=(300) 4007 &1  ; #4模组右边状态
OUT TR0
AND T0095  ; #4模组右电池感应屏蔽
AND H33.04  ; #4模组放料完成
AND H33.01  ; #4模组右有料
ANDNOT H33.02  ; #4模组测试完成
ANDNOT H0.03  ; #4模组屏蔽
AND W19.10  ; 启动状态
MOV(021) &2 4007  ; #4模组右边状态
LD TR0
AND T0094  ; #4模组左电池感应屏蔽
AND H33.04  ; #4模组放料完成
AND H33.00  ; #4模组左有料
ANDNOT H33.01  ; #4模组右有料
ANDNOT H33.02  ; #4模组测试完成
ANDNOT H0.03  ; #4模组屏蔽
AND W19.10  ; 启动状态
MOV(021) &3 4007  ; #4模组右边状态
; rung 10: #4模组左有料，左夹料气缸输出
LD=(300) 4006 &2  ; #4模组左边状态
AND W19.10  ; 启动状态
@SET W33.00  ; #4左夹料气缸输出
AND T0053  ; #4左夹料气缸夹紧位时间
MOV(021) &4 4006  ; #4模组左边状态
; rung 11: #4模组左有料状态下左密封气缸伸出
LD=(300) 4006 &4  ; #4模组左边状态
@SET W33.03  ; #4左密封气缸输出
AND T0049  ; #4左密封气缸伸出位时间
LDNOT 4.03  ; #4检漏仪Busy信号
OR P_On
ANDLD
MOV(021) &6 4006  ; #4模组左边状态

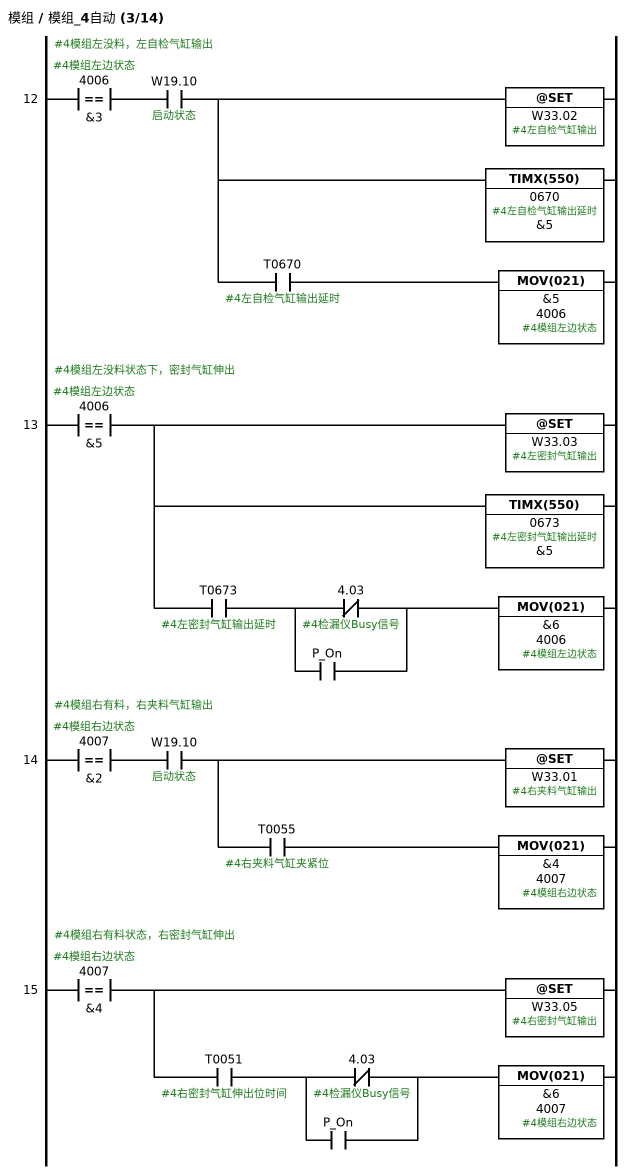
; rung 12: #4模组左没料，左自检气缸输出
LD=(300) 4006 &3  ; #4模组左边状态
AND W19.10  ; 启动状态
@SET W33.02  ; #4左自检气缸输出
TIMX(550) 0670 &5  ; #4左自检气缸输出延时
AND T0670  ; #4左自检气缸输出延时
MOV(021) &5 4006  ; #4模组左边状态
; rung 13: #4模组左没料状态下，密封气缸伸出
LD=(300) 4006 &5  ; #4模组左边状态
@SET W33.03  ; #4左密封气缸输出
TIMX(550) 0673 &5  ; #4左密封气缸输出延时
AND T0673  ; #4左密封气缸输出延时
LDNOT 4.03  ; #4检漏仪Busy信号
OR P_On
ANDLD
MOV(021) &6 4006  ; #4模组左边状态
; rung 14: #4模组右有料，右夹料气缸输出
LD=(300) 4007 &2  ; #4模组右边状态
AND W19.10  ; 启动状态
@SET W33.01  ; #4右夹料气缸输出
AND T0055  ; #4右夹料气缸夹紧位
MOV(021) &4 4007  ; #4模组右边状态
; rung 15: #4模组右有料状态，右密封气缸伸出
LD=(300) 4007 &4  ; #4模组右边状态
@SET W33.05  ; #4右密封气缸输出
AND T0051  ; #4右密封气缸伸出位时间
LDNOT 4.03  ; #4检漏仪Busy信号
OR P_On
ANDLD
MOV(021) &6 4007  ; #4模组右边状态

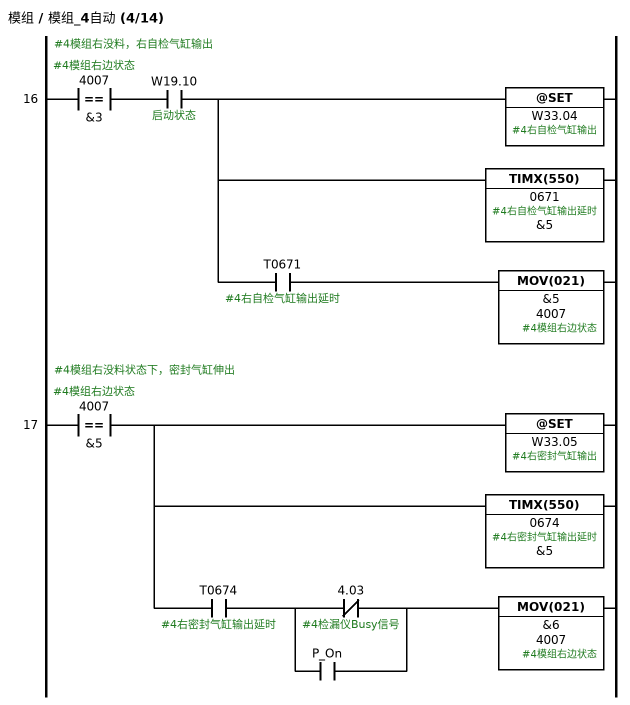
; rung 16: #4模组右没料，右自检气缸输出
LD=(300) 4007 &3  ; #4模组右边状态
AND W19.10  ; 启动状态
@SET W33.04  ; #4右自检气缸输出
TIMX(550) 0671 &5  ; #4右自检气缸输出延时
AND T0671  ; #4右自检气缸输出延时
MOV(021) &5 4007  ; #4模组右边状态
; rung 17: #4模组右没料状态下，密封气缸伸出
LD=(300) 4007 &5  ; #4模组右边状态
@SET W33.05  ; #4右密封气缸输出
TIMX(550) 0674 &5  ; #4右密封气缸输出延时
AND T0674  ; #4右密封气缸输出延时
LDNOT 4.03  ; #4检漏仪Busy信号
OR P_On
ANDLD
MOV(021) &6 4007  ; #4模组右边状态

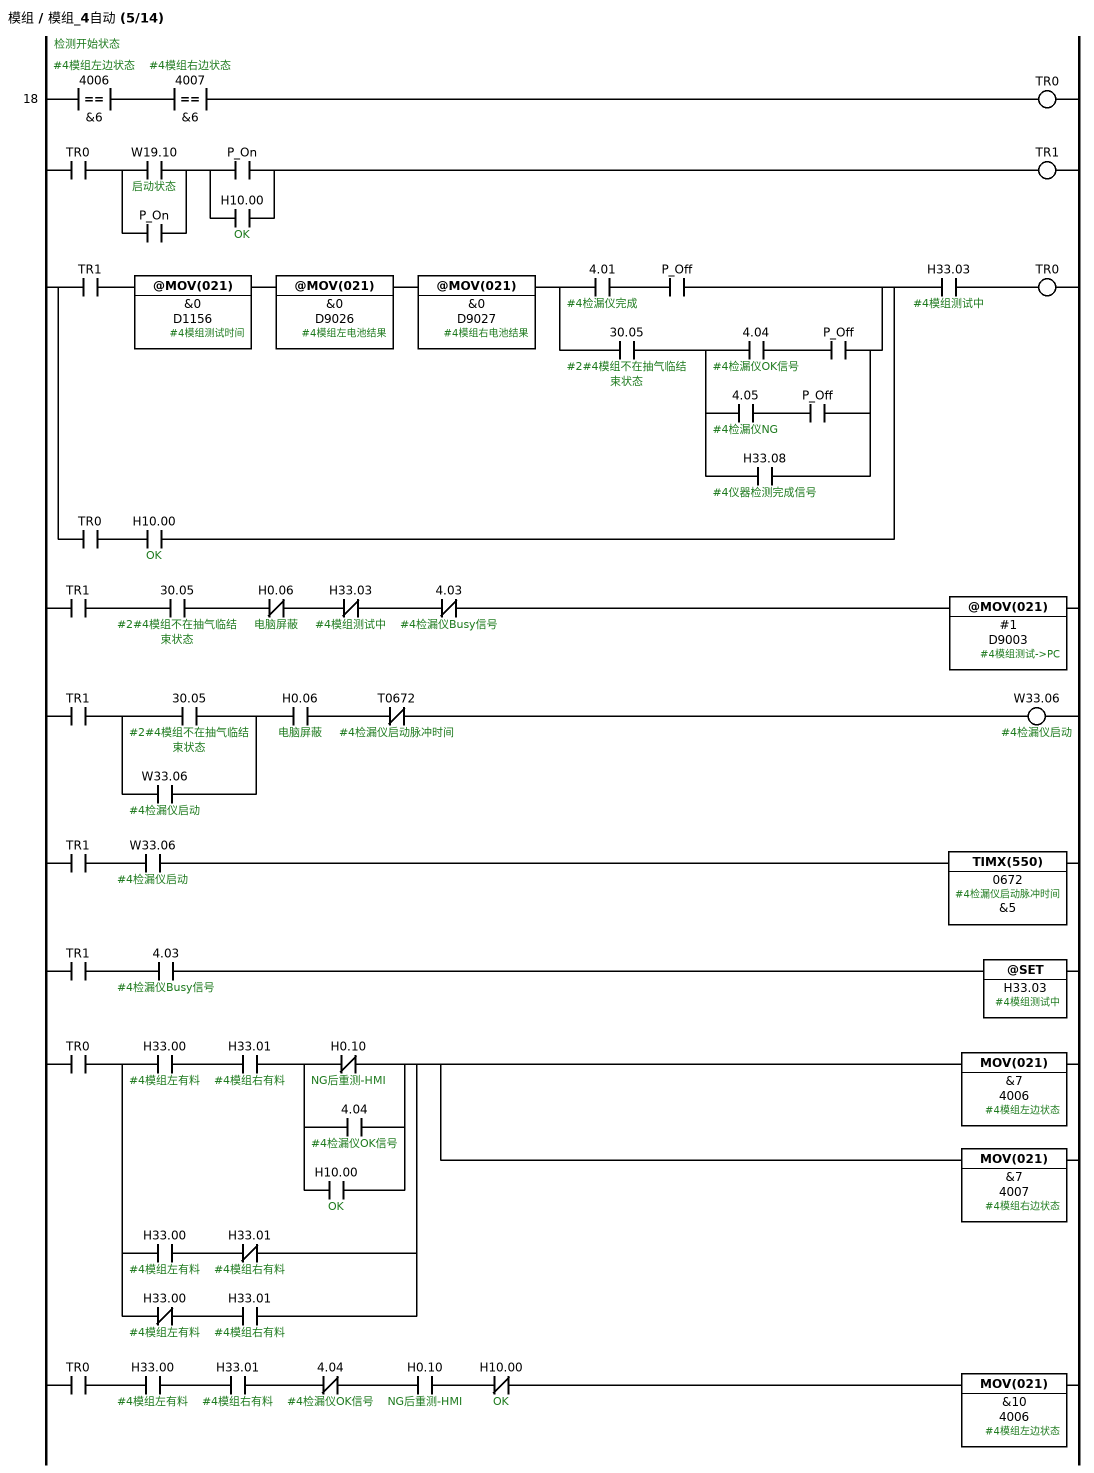
; rung 18: 检测开始状态
LD=(300) 4006 &6  ; #4模组左边状态
AND=(300) 4007 &6  ; #4模组右边状态
OUT TR0
LD W19.10  ; 启动状态
OR P_On
ANDLD
LD P_On  // 2018/5/28hy修改 所有模组不在抽气临结束状态下，下一模组才能启动(防抽气NG)
OR H10.00  ; OK
ANDLD
OUT TR1
AND 30.05  ; #2#4模组不在抽气临结束状态  // 2018/5/28hy修改 所有模组不在抽气临结束状态下，下一模组才能启动(防抽气NG)
ANDNOT H0.06  ; 电脑屏蔽
ANDNOT H33.03  ; #4模组测试中
ANDNOT 4.03  ; #4检漏仪Busy信号
@MOV(021) #1 D9003  ; #4模组测试->PC
LD TR1
LD 30.05  ; #2#4模组不在抽气临结束状态  // 2018/5/28hy修改 所有模组不在抽气临结束状态下，下一模组才能启动(防抽气NG)
OR W33.06  ; #4检漏仪启动
ANDLD
AND H0.06  ; 电脑屏蔽
ANDNOT T0672  ; #4检漏仪启动脉冲时间
OUT W33.06  ; #4检漏仪启动
LD TR1
AND W33.06  ; #4检漏仪启动
TIMX(550) 0672 &5  ; #4检漏仪启动脉冲时间
LD TR1
AND 4.03  ; #4检漏仪Busy信号
@SET H33.03  ; #4模组测试中
LD TR1
@MOV(021) &0 D1156  ; #4模组测试时间
@MOV(021) &0 D9026  ; #4模组左电池结果
@MOV(021) &0 D9027  ; #4模组右电池结果
LD 4.01  ; #4检漏仪完成
AND P_Off
LD 30.05  ; #2#4模组不在抽气临结束状态  // 2018/5/29hy修改,所有模组不在临抽气结束状态下，测试模组测试完成后，给出停止测试信号
LD 4.04  ; #4检漏仪OK信号
AND P_Off
LD 4.05  ; #4检漏仪NG
AND P_Off
ORLD
OR H33.08  ; #4仪器检测完成信号
ANDLD
ORLD
ANDLD
LD TR0
AND H10.00  ; OK
ORLD
AND H33.03  ; #4模组测试中
OUT TR0
LD H33.00  ; #4模组左有料
AND H33.01  ; #4模组右有料
LDNOT H0.10  ; NG后重测-HMI
OR 4.04  ; #4检漏仪OK信号
OR H10.00  ; OK
ANDLD
LD H33.00  ; #4模组左有料
ANDNOT H33.01  ; #4模组右有料
ORLD
LDNOT H33.00  ; #4模组左有料
AND H33.01  ; #4模组右有料
ORLD
ANDLD
MOV(021) &7 4006  ; #4模组左边状态
MOV(021) &7 4007  ; #4模组右边状态
LD TR0
AND H33.00  ; #4模组左有料
AND H33.01  ; #4模组右有料
ANDNOT 4.04  ; #4检漏仪OK信号
AND H0.10  ; NG后重测-HMI
ANDNOT H10.00  ; OK
MOV(021) &10 4006  ; #4模组左边状态

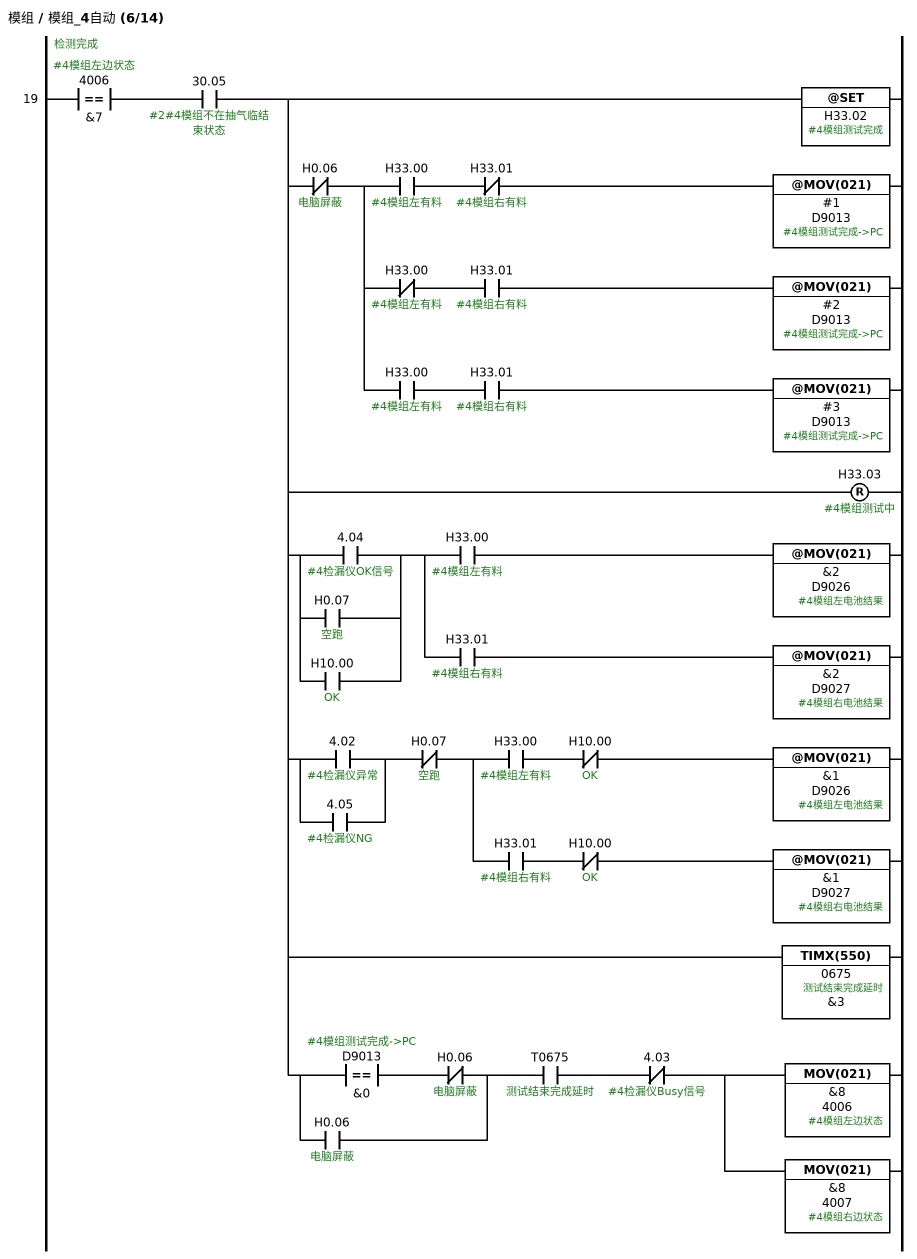
; rung 19: 检测完成
LD=(300) 4006 &7  ; #4模组左边状态
AND 30.05  ; #2#4模组不在抽气临结束状态
OUT TR0
@SET H33.02  ; #4模组测试完成
ANDNOT H0.06  ; 电脑屏蔽
OUT TR1
AND H33.00  ; #4模组左有料
ANDNOT H33.01  ; #4模组右有料
@MOV(021) #1 D9013  ; #4模组测试完成->PC
LD TR1
ANDNOT H33.00  ; #4模组左有料
AND H33.01  ; #4模组右有料
@MOV(021) #2 D9013  ; #4模组测试完成->PC
LD TR1
AND H33.00  ; #4模组左有料
AND H33.01  ; #4模组右有料
@MOV(021) #3 D9013  ; #4模组测试完成->PC
LD TR0
RSET H33.03  ; #4模组测试中
LD 4.04  ; #4检漏仪OK信号
OR H0.07  ; 空跑
OR H10.00  ; OK
ANDLD
OUT TR1
AND H33.00  ; #4模组左有料
@MOV(021) &2 D9026  ; #4模组左电池结果
LD TR1
AND H33.01  ; #4模组右有料
@MOV(021) &2 D9027  ; #4模组右电池结果
LD TR0
LD 4.02  ; #4检漏仪异常
OR 4.05  ; #4检漏仪NG
ANDLD
ANDNOT H0.07  ; 空跑
OUT TR1
AND H33.00  ; #4模组左有料
ANDNOT H10.00  ; OK
@MOV(021) &1 D9026  ; #4模组左电池结果
LD TR1
AND H33.01  ; #4模组右有料
ANDNOT H10.00  ; OK
@MOV(021) &1 D9027  ; #4模组右电池结果
LD TR0
TIMX(550) 0675 &3  ; 测试结束完成延时
LD=(300) D9013 &0  ; #4模组测试完成->PC
ANDNOT H0.06  ; 电脑屏蔽
OR H0.06  ; 电脑屏蔽
ANDLD
AND T0675  ; 测试结束完成延时
ANDNOT 4.03  ; #4检漏仪Busy信号
MOV(021) &8 4006  ; #4模组左边状态
MOV(021) &8 4007  ; #4模组右边状态

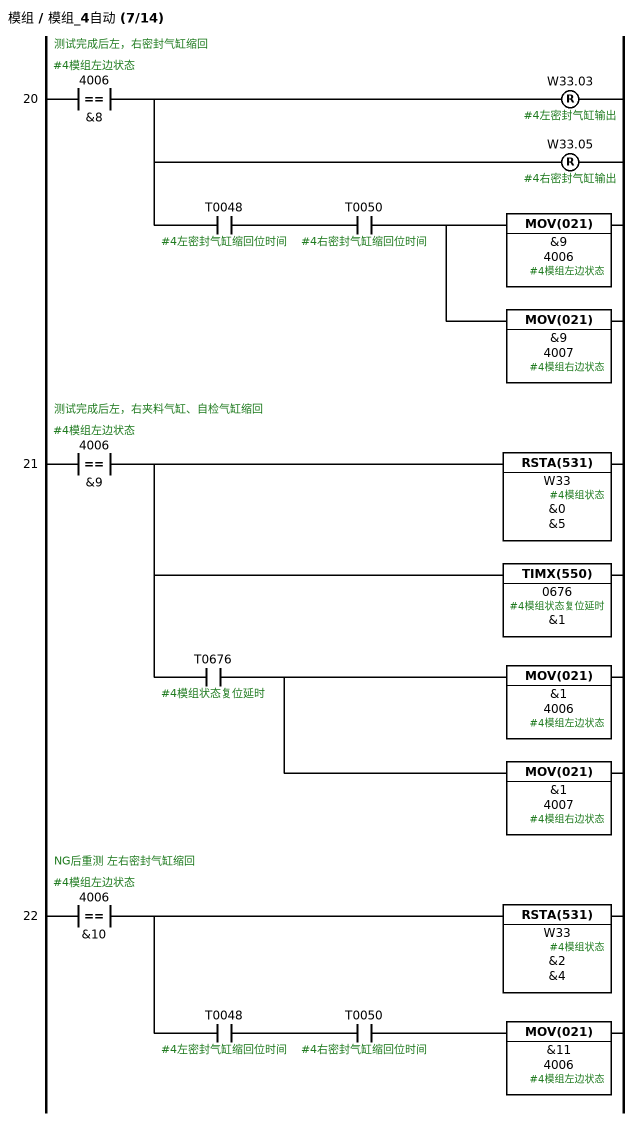
; rung 20: 测试完成后左，右密封气缸缩回
LD=(300) 4006 &8  ; #4模组左边状态
RSET W33.03  ; #4左密封气缸输出
RSET W33.05  ; #4右密封气缸输出
AND T0048  ; #4左密封气缸缩回位时间
AND T0050  ; #4右密封气缸缩回位时间
MOV(021) &9 4006  ; #4模组左边状态
MOV(021) &9 4007  ; #4模组右边状态
; rung 21: 测试完成后左，右夹料气缸、自检气缸缩回
LD=(300) 4006 &9  ; #4模组左边状态
RSTA(531) W33 &0 &5  ; #4模组状态
TIMX(550) 0676 &1  ; #4模组状态复位延时
AND T0676  ; #4模组状态复位延时
MOV(021) &1 4006  ; #4模组左边状态
MOV(021) &1 4007  ; #4模组右边状态
; rung 22: NG后重测 左右密封气缸缩回
LD=(300) 4006 &10  ; #4模组左边状态
RSTA(531) W33 &2 &4  ; #4模组状态
AND T0048  ; #4左密封气缸缩回位时间
AND T0050  ; #4右密封气缸缩回位时间
MOV(021) &11 4006  ; #4模组左边状态

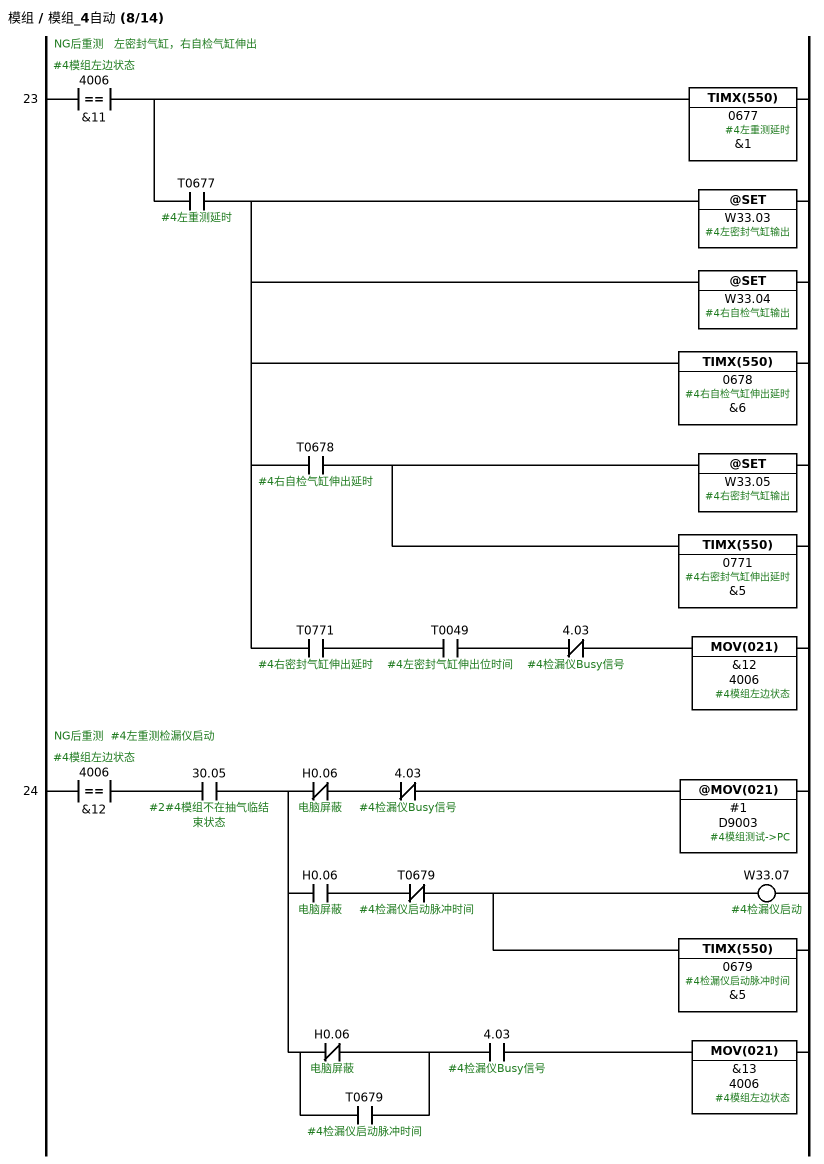
; rung 23: NG后重测   左密封气缸，右自检气缸伸出
LD=(300) 4006 &11  ; #4模组左边状态
TIMX(550) 0677 &1  ; #4左重测延时
AND T0677  ; #4左重测延时
OUT TR0
@SET W33.03  ; #4左密封气缸输出
@SET W33.04  ; #4右自检气缸输出
TIMX(550) 0678 &6  ; #4右自检气缸伸出延时
AND T0678  ; #4右自检气缸伸出延时
@SET W33.05  ; #4右密封气缸输出
TIMX(550) 0771 &5  ; #4右密封气缸伸出延时
LD TR0
AND T0771  ; #4右密封气缸伸出延时
AND T0049  ; #4左密封气缸伸出位时间
ANDNOT 4.03  ; #4检漏仪Busy信号
MOV(021) &12 4006  ; #4模组左边状态
; rung 24: NG后重测  #4左重测检漏仪启动
LD=(300) 4006 &12  ; #4模组左边状态
AND 30.05  ; #2#4模组不在抽气临结束状态  // 2018/5/28hy修改 所有模组不在抽气临结束状态下，下一模组才能启动(防抽气NG)
OUT TR0
ANDNOT H0.06  ; 电脑屏蔽
ANDNOT 4.03  ; #4检漏仪Busy信号
@MOV(021) #1 D9003  ; #4模组测试->PC
LD TR0
AND H0.06  ; 电脑屏蔽
ANDNOT T0679  ; #4检漏仪启动脉冲时间
OUT W33.07  ; #4检漏仪启动
TIMX(550) 0679 &5  ; #4检漏仪启动脉冲时间
LD TR0
LDNOT H0.06  ; 电脑屏蔽
OR T0679  ; #4检漏仪启动脉冲时间
ANDLD
AND 4.03  ; #4检漏仪Busy信号
MOV(021) &13 4006  ; #4模组左边状态

